VAR_GLOBAL
	nHomingError:UDINT:=16#14D00;
	axes			:	ARRAY [1..GVL.axisNum] OF AxisStruct;	//Global array of axisControl structure for holding axis parameters and controls
	//indexer			:	ARRAY [1..GVL.axisNum] OF IndexerStruct;
	
END_VAR

VAR_GLOBAL CONSTANT
	axisNum	:	UINT:=1;
	//axisCoupleMax	:	UINT:=4;
END_VAR

(* stored: Version 1.1.0.1, ProductVersion 3.1.4022.17
   GVL GVL: Id {913e21aa-a47e-444c-bfce-679b16c0434b} *)
